Yaskawa INFORM job: trapez_21_12_2023_planes_program.JBI

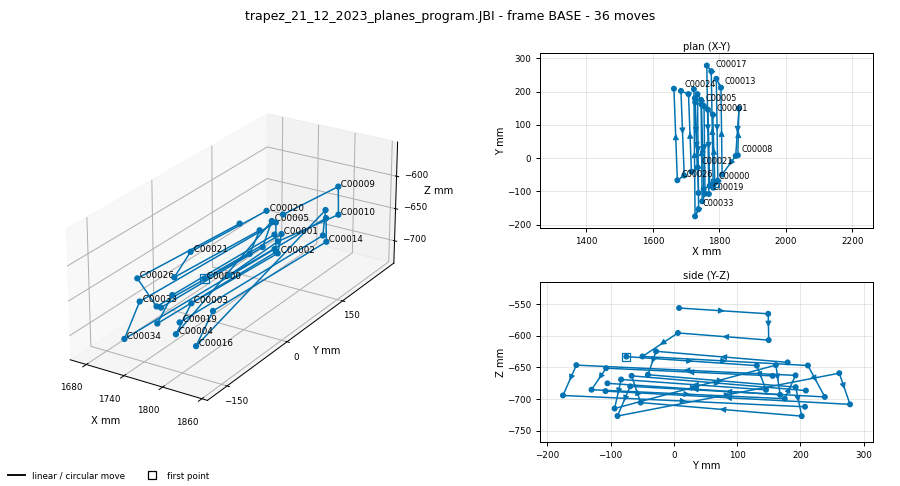
[picture p0: tool path of trapez_21_12_2023_planes_program.JBI in frame BASE, 36 of 41 moves have a stored position in this frame; points joined in program order, loops and branches not executed]
/JOB
//NAME trapez_21_12_2023_planes_program
//POS
///NPOS 36,0,36,0,0,0
///TOOL 0
///POSTYPE BASE
///RECTAN
///RCONF 0,0,0,0,0,0,0,0,0,0,0,0,0,0,0,0,0,0,0,0,0,0,0,0
C00000=1786.351931,-75.064449,-633.021071,175.000000,-68.670129,-5.000000
C00001=1780.136150,131.151880,-647.237451,175.000000,-68.670129,-5.000000
C00002=1765.637245,145.700875,-685.534618,175.000000,-68.670129,-5.000000
C00003=1770.978889,-83.349371,-669.133989,175.000000,-68.670129,-5.000000
C00004=1752.715941,-93.600865,-715.003450,175.000000,-68.670129,-5.000000
C00005=1746.206916,161.328661,-646.434390,175.000000,-68.670129,-5.000000
C00006=1727.241055,167.935828,-693.390022,175.000000,-68.670129,-5.000000
C00007=1737.116796,-104.949166,-675.222021,180.000000,-60.000000,0.000000
C00008=1855.621716,8.328367,-556.190803,175.000000,-73.990827,-5.000000
C00009=1858.622481,149.198597,-565.325825,175.000000,-73.990827,-5.000000
C00010=1859.264372,149.972573,-606.954672,175.000000,-73.990827,-5.000000
C00011=1849.092803,6.514885,-595.610251,175.000000,-73.990827,-5.000000
C00012=1808.329171,-49.532273,-632.722668,175.000000,-73.990827,-5.000000
C00013=1804.761515,211.917163,-647.055317,175.000000,-73.990827,-5.000000
C00014=1790.825516,238.657161,-696.727592,175.000000,-73.990827,-5.000000
C00015=1795.463065,-68.935938,-679.991659,175.000000,-73.990827,-5.000000
C00016=1781.475334,-89.098016,-726.894290,175.000000,-73.990827,-5.000000
C00017=1775.592600,261.493699,-659.195947,175.000000,-73.990827,-5.000000
C00018=1762.224072,278.486295,-708.458525,175.000000,-73.990827,-5.000000
C00019=1768.492581,-108.004204,-687.556493,180.000000,-60.000000,0.000000
C00020=1726.131041,179.906623,-642.104324,-175.000000,-64.089664,-5.000000
C00021=1734.128599,-28.125941,-624.622331,-175.000000,-64.089664,-5.000000
C00022=1715.948295,-40.927949,-661.582220,-175.000000,-64.089664,-5.000000
C00023=1707.085696,192.637622,-681.266499,-175.000000,-64.089664,-5.000000
C00024=1684.457541,202.134768,-727.073731,-175.000000,-64.089664,-5.000000
C00025=1694.232697,-52.427849,-705.676146,-175.000000,-64.089664,-5.000000
C00026=1673.608381,-66.729919,-663.409860,-175.000000,-64.089664,-5.000000
C00027=1663.313506,208.766752,-686.705120,180.000000,-60.000000,0.000000
C00028=1753.813130,156.174697,-663.468596,175.000000,-76.523357,5.000000
C00029=1756.903329,-107.071927,-651.291089,175.000000,-76.523357,5.000000
C00030=1748.150130,-130.090231,-685.323049,175.000000,-76.523357,5.000000
C00031=1744.946982,175.291222,-699.541130,175.000000,-76.523357,5.000000
C00032=1734.240801,192.368369,-662.685133,175.000000,-76.523357,5.000000
C00033=1737.531906,-154.113690,-646.471237,175.000000,-76.523357,5.000000
C00034=1726.906209,-175.218112,-694.363418,175.000000,-76.523357,5.000000
C00035=1723.371787,207.261827,-712.285495,180.000000,-60.000000,0.000000
///POSTYPE PULSE
///PULSE
EC00000=23552.0
EC00001=23552.0
EC00002=23552.0
EC00003=23552.0
EC00004=23552.0
EC00005=23552.0
EC00006=23552.0
EC00007=23552.0
EC00008=115712.0
EC00009=115712.0
EC00010=115712.0
EC00011=115712.0
EC00012=115712.0
EC00013=115712.0
EC00014=115712.0
EC00015=115712.0
EC00016=115712.0
EC00017=115712.0
EC00018=115712.0
EC00019=115712.0
EC00020=207872.0
EC00021=207872.0
EC00022=207872.0
EC00023=207872.0
EC00024=207872.0
EC00025=207872.0
EC00026=207872.0
EC00027=207872.0
EC00028=300032.0
EC00029=300032.0
EC00030=300032.0
EC00031=300032.0
EC00032=300032.0
EC00033=300032.0
EC00034=300032.0
EC00035=300032.0
//INST
///DATE 2023/07/21 14:02
///ATTR SC,RW,RJ
////FRAME BASE
///GROUP1 RB1,ST1
NOP
MOVJ P009 EX000 VJ=15.00
MOVJ C00000 EC00000 VJ=15.0
MOVL C00001 EC00001 V=150.0
MOVL C00002 EC00002 V=150.0
MOVL C00003 EC00003 V=150.0
MOVL C00004 EC00004 V=150.0
MOVL C00005 EC00005 V=150.0
MOVL C00006 EC00006 V=150.0
MOVL C00007 EC00007 V=150.0
MOVJ P009 VJ=15.00
MOVJ C00008 EC00008 VJ=15.0
MOVL C00009 EC00009 V=150.0
MOVL C00010 EC00010 V=150.0
MOVL C00011 EC00011 V=150.0
MOVL C00012 EC00012 V=150.0
MOVL C00013 EC00013 V=150.0
MOVL C00014 EC00014 V=150.0
MOVL C00015 EC00015 V=150.0
MOVL C00016 EC00016 V=150.0
MOVL C00017 EC00017 V=150.0
MOVL C00018 EC00018 V=150.0
MOVL C00019 EC00019 V=150.0
MOVJ P009 VJ=15.00
MOVJ C00020 EC00020 VJ=15.0
MOVL C00021 EC00021 V=150.0
MOVL C00022 EC00022 V=150.0
MOVL C00023 EC00023 V=150.0
MOVL C00024 EC00024 V=150.0
MOVL C00025 EC00025 V=150.0
MOVL C00026 EC00026 V=150.0
MOVL C00027 EC00027 V=150.0
MOVJ P009 VJ=15.00
MOVJ C00028 EC00028 VJ=15.0
MOVL C00029 EC00029 V=150.0
MOVL C00030 EC00030 V=150.0
MOVL C00031 EC00031 V=150.0
MOVL C00032 EC00032 V=150.0
MOVL C00033 EC00033 V=150.0
MOVL C00034 EC00034 V=150.0
MOVL C00035 EC00035 V=150.0
MOVJ P009 VJ=15.00
END
